FUNCTION_BLOCK FB_TestSuiteWithClock EXTENDS TcUnit.FB_TestSuite

METHOD PROTECTED AdvanceClockMs
VAR_INPUT
	Duration : TIME;
END_VAR
// No Op; xSTunit compatibility adapter.
END_METHOD

METHOD PROTECTED AdvanceClockNs
VAR_INPUT
	Duration : LTIME;
END_VAR
// No Op; xSTunit compatibility adapter.
END_METHOD

END_FUNCTION_BLOCK

(* stored: Version 1.1.0.1, ProductVersion 3.1.4026.18
   POU FB_TestSuiteWithClock: Id {267d7f54-cead-459f-9b43-6ee4e810c1a1}, SpecialFunc None
   Method AdvanceClockMs: Id {4a5b9e20-07bf-4e8f-bdf8-7f689e559b77}
   Method AdvanceClockNs: Id {472b7be4-8c4e-4d86-959f-59c18551dcbb} *)
